// Mitsubishi GX Works2 project: 240507_timechart13_ctr링카운터2gxw   PLC: Q03UDV

PROGRAM MAIN
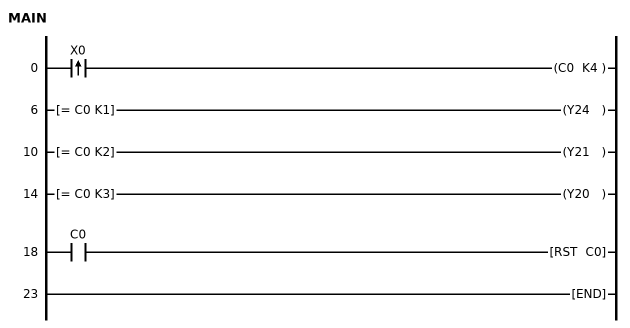
0     LDP     X0
      OUT     C0 K4
6     LD=     C0 K1
      OUT     Y24
10    LD=     C0 K2
      OUT     Y21
14    LD=     C0 K3
      OUT     Y20
18    LD      C0
      RST     C0
23    END
END_PROGRAM
